FUNCTION F_CAMERA_LightingIntensity : INT
VAR_INPUT
	nUnitLightingIntensity		:INT;
END_VAR

F_CAMERA_LightingIntensity := LREAL_TO_INT(LIMIT(0, INT_TO_LREAL(nUnitLightingIntensity), 100)*32767.0/100);

END_FUNCTION

(* stored: Version 1.1.0.1
   POU F_CAMERA_LightingIntensity: Id {d2762582-2f5a-4092-a8f1-5b04be1e67bd}, SpecialFunc None *)
